VAR_GLOBAL

//******************** Strona I ********************  
	bCompressedAirFlowImpulse AT %I* : BOOL;		// Impuls co 30L
	bCompressedAirFlowAlarmHigh AT %I* : BOOL;		// Alarm gdy przekroczony przepływ 300L/min
	bCompressedAirFlowImpulsePreAssembly			AT %I* :BOOL;
	bCompressedAirFlowImpulseFilling	 			AT %I* :BOOL;
	bCompressedAirFlowImpulseHotPlate	 			AT %I* :BOOL;
// Komunikacja RS485
// S01
	stS01_1_BearingPress_IO				: stSonicPress_DigInOuts_V4_1;
	bS01_Trigger			 			AT %Q* :BOOL;
	bS01_Result 						AT %I* :BOOL;
	bS01_Ready	 						AT %I* :BOOL;
	
// S02	- 
	stS02_1_BearingPress_IO				: stSonicPress_DigInOuts_V4_1;
	
// S03 - 
	stS03_1_BearingPress_IO				: stSonicPress_DigInOuts_V4_1;
	stS03_CapFixture_IO					: stCapDetectionInOuts;
// S04 - 
	stS04_1_BearingPress_IO				: stSonicPress_DigInOuts_V4_1;
	
	
// Sxx Plug A - 
	stSxxA_1_PlugAWelder_IO				: stSonicTech_DigInOuts_V3_1;
	
	
// Sxx Plug B - 
	stSxxB_1_PlugAWelder_IO				: stSonicTech_DigInOuts_V3_1;
//	Bottle filling line
		//S02
	b_1_SonicTech_EnergyConsumptionImp 				AT %I* :BOOL;
	st_1_SonicTech_WeldingMachine_IO				: stSonicTech_DigInOuts_V4_1;
	//S04
	b_2_SonicTech_EnergyConsumptionImp 				AT %I* :BOOL;
	st_2_SonicTech_WeldingMachine_IO				: stSonicTech_DigInOuts_V4_1;
	//S05
	stUnderPreserInOuts 							: stUnderPressureTesterInOuts_V3_1;
	stTransporterInOuts								: stTransporterInOuts_V3_2;
	stUnderPressureInOuts_V2						: stUnderPressureTesterInOuts_V3_1;
	//S07
	stTunelInOuts									: stDetectionTunelInOuts_V3_1;
	stSerialData_S02_S04 				: stSerialComData;
END_VAR

(* stored: Version 1.1.0.1, ProductVersion 3.1.4024.15
   GVL GVL_IO: Id {3a3e8a3f-c558-4d33-83cd-786f8332bedc} *)
